PROGRAM LOGGING
VAR_INPUT
	sWriteLog		: STRING[255];
	sLog			: STRING[255];
//	dir_log 		: UINT;
	bLogFlag		: BOOL;
	LogState		: INT;
END_VAR
VAR_OUTPUT
	bError				: BOOL;
	nErrID				: UDINT;
END_VAR
VAR
	CreateDir	: FB_CreateDir;
	FileOpen	: FB_FileOpen;
	FileWrite	: FB_FileWrite;
	FileClose	: FB_FileClose;
	
    ePath        	: E_OpenPath; (* folders root path *)
    sPathName     	: STRING;
	bBootFolder		: BOOL;
	writeBuffer		: STRING[255] := '';
	hfile			: UINT;
	
	sTxtName	: T_MaxString;
	sFolderName	: T_MaxString;
	DirCreateError	: BOOL;
	FileOpenError	: BOOL;
	FileWriteError	: BOOL;
	FileCloseError	: BOOL;
	sTimeStamp: STRING(255);
	
	writeFlag		: BOOL;
	lastLog			: String[255];
END_VAR

IF sLog = lastLog THEN
	RETURN;
END_IF

//CASE LogState OF
//	0:
//		writeFlag := TRUE;
//		// Set Log Folder Name
////		sFolderName := CONCAT ('C:\Users\celli\OneDrive\Desktop\YISB_LOG\',LOG_TIME_STAMP.Local_Date);
//		sFolderName := CONCAT ('C:\Users\Administrator\Desktop\log\',LOG_TIME_STAMP.Local_Date);
		
//		CreateDir(
//				sNetId:= '', 
//				sPathName:= sFolderName, 
//				ePath:= PATH_GENERIC, 
//				bExecute:= TRUE, 
//				tTimeout:= DEFAULT_ADS_TIMEOUT, 
//				bBusy=> , 
//				bError=> DirCreateError, 
//				nErrId=> nErrID);
//			IF CreateDir.tTimeout > DEFAULT_ADS_TIMEOUT THEN
//				LogState := 0;
//				bLogFlag := FALSE;
//				CreateDir.bExecute := FALSE;
//				FileOpen(bExecute := FALSE);
//				MAIN.BTN_LOG := FALSE;
//				RETURN;
//			ELSIF NOT CreateDir.bBusy THEN
//				LogState := 1;
//				CreateDir.bExecute := FALSE;
//				FileOpen(bExecute := FALSE);
//			END_IF

//		// Open File	
//		1:
//			// Set Log File Name	
//			sTxtName := WORD_TO_STRING(LOG_TIME_STAMP.LocalTime.systemTime.wHour);
//			sTxtName := CONCAT(sTxtName, '.txt');
//			sTxtName := CONCAT('\',sTxtName,);
//			sTxtName := CONCAT(sFolderName,sTxtName);
			
//			FileOpen(
//				sNetId:= , 
//				sPathName:= sTxtName, 
//				nMode:= FOPEN_MODEAPPEND, 
//				ePath:= PATH_GENERIC, 
//				bExecute:= TRUE, 
//				tTimeout:= DEFAULT_ADS_TIMEOUT, 
//				bBusy=> , 
//				bError=> FileOpenError, 
//				nErrId=> nErrID, 
//				hFile=> hfile);
//			IF FileOpenError OR FileOpen.tTimeout > DEFAULT_ADS_TIMEOUT THEN
//				LogState := 0;
//				bLogFlag := FALSE;
//				FileOpen.bExecute := FALSE;
//				FileWrite(bExecute := FALSE);
//				MAIN.BTN_LOG := FALSE;
//				RETURN;
//			ELSIF NOT FileOpen.bBusy THEN
//				LogState := 2;
//				FileOpen.bExecute := FALSE;
//				FileWrite(bExecute := FALSE);
//			END_IF
			
//		// Write File
//		2:	
//				// Set Log messages	
//				sTimeStamp 	:= CONCAT('$n',SYSTEMTIME_TO_STRING(LOG_TIME_STAMP.LocalTime.systemTime));
//				sTimeStamp 	:= CONCAT(sTimeStamp,' - ');
//				sWriteLog 	:= CONCAT(sTimeStamp, sLog);
//				writeBuffer := sWriteLog;
				
//				FileWrite(
//					sNetId:= , 
//					hFile:= hfile, 
//					pWriteBuff:= ADR(writeBuffer), 
//					cbWriteLen:= INT_TO_UDINT(LEN(writeBuffer)), 
//					bExecute:= TRUE, 
//					tTimeout:= T#3S, 
//					bBusy=> , 
//					bError=> FileWriteError, 
//					nErrId=> nErrID, 
//					cbWrite=> );
					
//			IF FileWriteError OR FileWrite.tTimeout > DEFAULT_ADS_TIMEOUT THEN
//				LogState := 0;
//				bLogFlag := FALSE;
//				FileWrite.bExecute := FALSE;
//				MAIN.BTN_LOG := FALSE;
//				writeFlag:= FALSE;
//				FileClose(bExecute := FALSE);
//				RETURN;
//			ELSIF NOT FileWrite.bBusy THEN
//				LogState := 3;
//				writeFlag:= FALSE;
//				FileWrite.bExecute := FALSE;
//				FileClose(bExecute := FALSE);
//			END_IF
			
//		// Close File
//		3:
//			FileClose(
//				sNetId:= , 
//				hFile:= hfile, 
//				bExecute:= TRUE,
//				tTimeout:= T#3S, 
//				bBusy=> , 
//				bError=> FileCloseError, 
//				nErrId=> nErrID);
//			IF FileCloseError OR FileClose.tTimeout > DEFAULT_ADS_TIMEOUT THEN
//				LogState := 0;
//				bLogFlag := FALSE;
//				lastLog := sLog;
//				FileClose(bExecute := FALSE);
//				MAIN.BTN_LOG := FALSE;
//				RETURN;
//			ELSIF NOT FileClose.bBusy THEN
//				LogState := 0;
//				lastLog := sLog;
//				FileClose(bExecute := FALSE);
//				CreateDir(bExecute:= FALSE);
//				bLogFlag := FALSE;
//				MAIN.BTN_LOG := FALSE;
//			END_IF
//END_CASE

END_PROGRAM

(* stored: Version 1.1.0.1, ProductVersion 3.1.4024.12
   POU LOGGING: Id {16605c93-8696-4973-a434-6ac70e0b45c2}, SpecialFunc None *)
